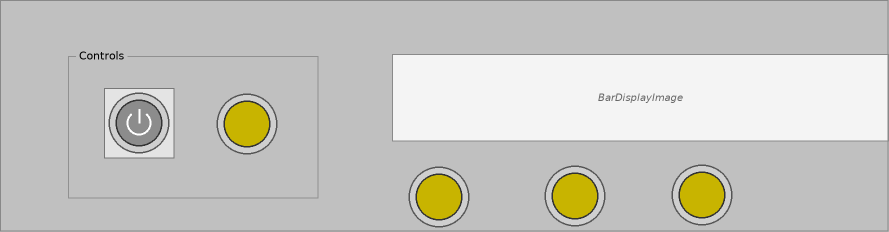
VISUALIZATION Visualization  // 889x232
    BarDisplayImage (392,54 497x87), value: PLC_TaskCase.stMachine1.fTemperature, style: BarDisplayImage-Gray, scale format: %.1f, scale 0..500
    GroupBox (68,48 250x150), "Controls"
        Lamp1 (144,41 70x70), variable: PLC_TaskCase.bStart, style: Lamp-Lamp1-Yellow
        PowerSwitch (36,40 70x70), variable: PLC_TaskCase.stMachine1.bStartButtonPressed, behaviour: TOGGLE, style: Switch-PowerSwitch-Gray
    Lamp1 (667,160 70x70), variable: PLC_TaskCase.stMachine1.bIsCooling, style: Lamp-Lamp1-Yellow
    Lamp1 (540,161 70x70), variable: PLC_TaskCase.stMachine1.bIsSmelting, style: Lamp-Lamp1-Yellow
    Lamp1 (404,162 70x70), variable: PLC_TaskCase.stMachine1.bIsHeating, style: Lamp-Lamp1-Yellow
END_VISUALIZATION

(* stored: Version 1.1.0.1, ProductVersion 3.1.4024.12
   Visu Visualization: Id {7c879211-aa37-4102-884c-b2d065071ef8} *)
